FUNCTION_BLOCK FB_TON (* standard timer function block (on-delay timing) *)
  (* Standard: 61131-3; Classification: standard timer function block *)
  (* Version 1.0, 2009-09-14, 4DIAC-IDE, 4DIAC-Consortium *)
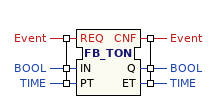
  EVENT_INPUT
    REQ WITH IN, PT; (* Normal Execution Request *)
  END_EVENT
  EVENT_OUTPUT
    CNF WITH Q, ET; (* Execution Confirmation *)
  END_EVENT
  VAR_INPUT
    IN : BOOL; (* Input *)
    PT : TIME; (* Process time *)
  END_VAR
  VAR_OUTPUT
    Q : BOOL; (* Output *)
    ET : TIME; (* Elapsed time *)
  END_VAR
END_FUNCTION_BLOCK
